// TIA Portal project "Cau4" (V16)

(* hardware
DEVICE "S7-1200 station_1"  S7-1200 Station
   slot 0: "Rack_0"  S7-1200 Rack  Rack  V1.0
   slot 1: "PLC_1"  CPU 1212C DC/DC/DC  6ES7 212-1AE40-0XB0  V4.3
   slot 2: "DI 16/DQ 16x24VDC_1"  6ES7 223-1BL32-0XB0  V2.0
   slot 3: "DQ 16xRelay_1"  SM 1222 DQ16 x relay  6ES7 222-1HH32-0XB0  V2.0
*)

// ===== PLC "PLC_1"  CPU 1212C DC/DC/DC =====

VAR_GLOBAL   // PLC tag table "Default tag table"
   "Stop" AT %I8.2 : Bool;
   "Start" AT %I8.3 : Bool;
   "Biến giữ chương trình" AT %M0.0 : Bool;
   "A/M" AT %I8.4 : Bool;
   "KM1" AT %Q0.0 : Bool;
   "KM2" AT %Q0.1 : Bool;
   "KM3" AT %Q0.2 : Bool;
   "KM4" AT %Q0.3 : Bool;
   "KM5" AT %Q0.4 : Bool;
   "B (NO)" AT %I0.6 : Bool;
   "C (NO)" AT %I0.7 : Bool;
   "Tag_4" AT %I1.0 : Bool;
   "Tag_5" AT %I1.1 : Bool;
   "Tag_6" AT %I0.1 : Bool;
   "Tag_7" AT %I0.2 : Bool;
   "Tag_8" AT %M0.1 : Bool;
   "Biến bật KM2" AT %M0.2 : Bool;
   "Biến bật KM3" AT %M0.3 : Bool;
   "Biến bật KM4" AT %M0.4 : Bool;
   "Biến bật KM5" AT %M0.5 : Bool;
   "A (NO)" AT %I0.5 : Bool;
   "D (NO)" AT %I8.0 : Bool;
END_VAR

// folder: System blocks/Program resources

DATA_BLOCK "T1"   // DB1
{ S7_Optimized_Access := 'TRUE' }
AUTHOR : Simatic
FAMILY : IEC
NAME : IEC_TMR
VERSION : 1.0
// stored: InstanceOfName IEC_TIMER
"IEC_TIMER"
BEGIN
END_DATA_BLOCK

// folder: (top level)

ORGANIZATION_BLOCK "Main"   // OB1, LAD, ProgramCycle
TITLE = "Main Program Sweep (Cycle)"
{ S7_Optimized_Access := 'TRUE' }
VERSION : 0.1
   VAR_INPUT
      Initial_Call : Bool;   // Initial call of this OB
      Remanence : Bool;   // =True, if remanent data are available
   END_VAR
BEGIN

REGION Network 1
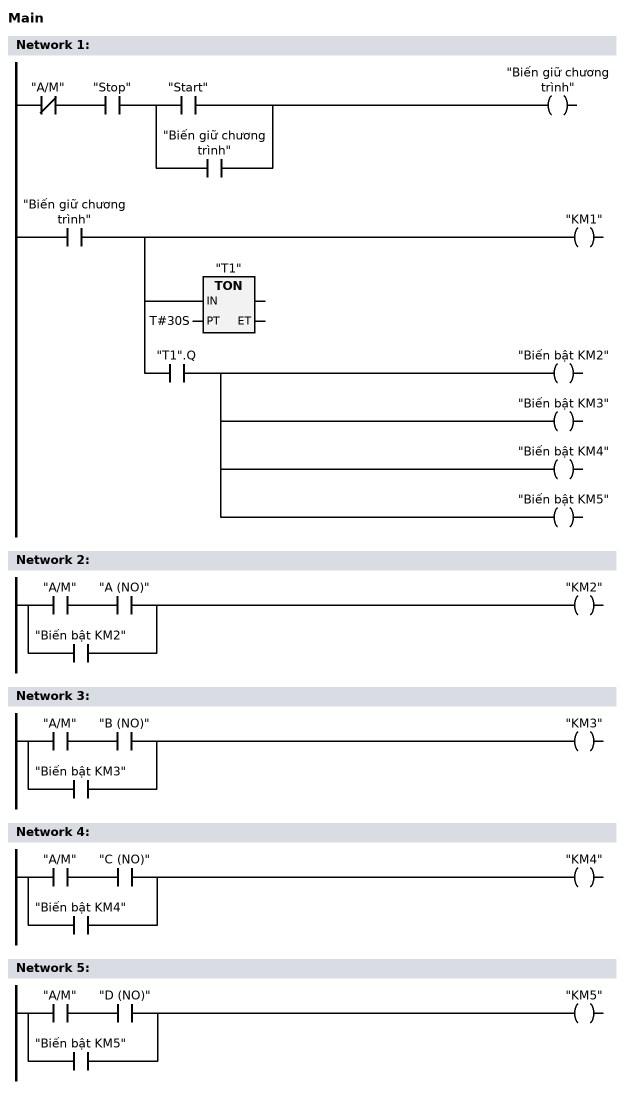
   "Biến giữ chương trình" := NOT "A/M" AND "Stop" AND ("Start" OR "Biến giữ chương trình");
   "KM1" := "Biến giữ chương trình";
   "T1".TON(IN := "Biến giữ chương trình", PT := T#30S);
   "Biến bật KM2" := "Biến giữ chương trình" AND "T1".Q;
   "Biến bật KM3" := "Biến bật KM2";
   "Biến bật KM4" := "Biến bật KM2";
   "Biến bật KM5" := "Biến bật KM2";
END_REGION

REGION Network 2
   RUNG wire#powerrail
      Contact( "A/M" )
      Contact( "A (NO)" )
      wire#w1
      Coil( "KM2" )
   END_RUNG
   RUNG wire#powerrail
      Contact( "Biến bật KM2" )
   END_RUNG wire#w1
   // the same network as SCL:
   "KM2" := ("A/M" AND "A (NO)") OR "Biến bật KM2";
END_REGION

REGION Network 3
   RUNG wire#powerrail
      Contact( "A/M" )
      Contact( "B (NO)" )
      wire#w1
      Coil( "KM3" )
   END_RUNG
   RUNG wire#powerrail
      Contact( "Biến bật KM3" )
   END_RUNG wire#w1
   // the same network as SCL:
   "KM3" := ("A/M" AND "B (NO)") OR "Biến bật KM3";
END_REGION

REGION Network 4
   RUNG wire#powerrail
      Contact( "A/M" )
      Contact( "C (NO)" )
      wire#w1
      Coil( "KM4" )
   END_RUNG
   RUNG wire#powerrail
      Contact( "Biến bật KM4" )
   END_RUNG wire#w1
   // the same network as SCL:
   "KM4" := ("A/M" AND "C (NO)") OR "Biến bật KM4";
END_REGION

REGION Network 5
   RUNG wire#powerrail
      Contact( "A/M" )
      Contact( "D (NO)" )
      wire#w1
      Coil( "KM5" )
   END_RUNG
   RUNG wire#powerrail
      Contact( "Biến bật KM5" )
   END_RUNG wire#w1
   // the same network as SCL:
   "KM5" := ("A/M" AND "D (NO)") OR "Biến bật KM5";
END_REGION
END_ORGANIZATION_BLOCK